// TwinCAT 3 PLC project SmartLogisticsBasic
// ProgramVersion: 3.1.4026.16
// libraries:
//   Tc2_BA, * (Beckhoff Automation GmbH)
//   Tc2_BABasic, * (Beckhoff Automation GmbH)
//   Tc2_BACnetRev12, * (Beckhoff Automation GmbH)
//   Tc2_CncBase, * (Beckhoff Automation GmbH)
//   Tc2_CncHli, * (Beckhoff Automation GmbH)
//   Tc2_CncPlcopenP1, * (Beckhoff Automation GmbH)
//   Tc2_CncPlcopenP4, * (Beckhoff Automation GmbH)
//   Tc2_ControllerToolbox, * (Beckhoff Automation GmbH)
//   Tc2_Coupler, * (Beckhoff Automation GmbH)
//   Tc2_DALI, * (Beckhoff Automation GmbH)
//   Tc2_Database, * (Beckhoff Automation GmbH)
//   Tc2_DataExchange, * (Beckhoff Automation GmbH)
//   Tc2_DMX, * (Beckhoff Automation GmbH)
//   Tc2_Drive, * (Beckhoff Automation GmbH)
//   Tc2_EIB, * (Beckhoff Automation GmbH)
//   Tc2_EnOcean, * (Beckhoff Automation GmbH)
//   Tc2_EtherCAT, * (Beckhoff Automation GmbH)
//   Tc2_EthernetIP, * (Beckhoff Automation GmbH)
//   Tc2_FTP, * (Beckhoff Automation GmbH)
//   Tc2_GENIbus, * (Beckhoff Automation GmbH)
//   Tc2_HVAC, * (Beckhoff Automation GmbH)
//   Tc2_IoFunctions, * (Beckhoff Automation GmbH)
//   Tc2_KL85xx, * (Beckhoff Automation GmbH)
//   Tc2_LON, * (Beckhoff Automation GmbH)
//   Tc2_Math, * (Beckhoff Automation GmbH)
//   Tc2_MBus, * (Beckhoff Automation GmbH)
//   Tc2_MC2, * (Beckhoff Automation GmbH)
//   Tc2_MC2_Camming, * (Beckhoff Automation GmbH)
//   Tc2_MC2_Drive, * (Beckhoff Automation GmbH)
//   Tc2_MC2_FlyingSaw, * (Beckhoff Automation GmbH)
//   Tc2_MC2_XFC, * (Beckhoff Automation GmbH)
//   Tc2_MDP, * (Beckhoff Automation GmbH)
//   Tc2_ModbusRTU, * (Beckhoff Automation GmbH)
//   Tc2_ModbusSrv, * (Beckhoff Automation GmbH)
//   Tc2_MPBus, * (Beckhoff Automation GmbH)
//   Tc2_NC, * (Beckhoff Automation GmbH)
//   Tc2_NcDrive, * (Beckhoff Automation GmbH)
//   Tc2_NcFifoAxes, * (Beckhoff Automation GmbH)
//   Tc2_NCI, * (Beckhoff Automation GmbH)
//   Tc2_NciXFC, * (Beckhoff Automation GmbH)
//   Tc2_PlcInterpolation, * (Beckhoff Automation GmbH)
//   Tc2_ProfinetDiag, * (Beckhoff Automation GmbH)
//   Tc2_RFID, * (Beckhoff Automation GmbH)
//   Tc2_S5S7Com, * (Beckhoff Automation GmbH)
//   Tc2_SerialCom, * (Beckhoff Automation GmbH)
//   Tc2_SMI, * (Beckhoff Automation GmbH)
//   Tc2_SMS, * (Beckhoff Automation GmbH)
//   Tc2_Smtp, * (Beckhoff Automation GmbH)
//   Tc2_SPA, * (Beckhoff Automation GmbH)
//   Tc2_Standard, * (Beckhoff Automation GmbH)
//   Tc2_System, * (Beckhoff Automation GmbH)
// project tree:
//   GVLs/ GVL_SimitSp.TcGVL, GVL_System.TcGVL (not stored)
//   / PlcTask.TcTTO
//   POUs/ FB_Chrono.TcPOU, FB_Conveyor.TcPOU (not stored), FB_ConvStatistic.TcPOU, FB_ConvSys.TcPOU, FB_FlPos.TcPOU, FB_MyUpCounter.TcPOU, FB_RunControl.TcPOU, FB_SpeedControl.TcPOU, FC_GetMaxLapTime.TcPOU, MAIN.TcPOU
// real-time tasks:
//   TASK PlcTask: cycle T#10ms, priority 20, ADS port 350
//   TASK OPC UA Virtual: cycle T#10ms, priority 35, ADS port 351
// I/O:
//   DEVICE Device 1 (OPC UA Virtual), AmsNetId 192.168.200.222.2.1
// variable links:
//   SmartLogisticsBasic Instance <-> Device 1 (OPC UA Virtual)/Siemens.Simit.OpcUaServer.OpcUaServerService
//     PlcTask Outputs/GVL_System.bWrite_Enable <-> Outputs/Control/Write Enable
//   SmartLogisticsBasic Instance <-> Device 1 (OPC UA Virtual)/Siemens.Simit.OpcUaServer.OpcUaServerService/urn:vmw11:Siemens:Simit.OpcUaServer.OPC UA Server/InSimitOpcBin/Ix_Enable
//     PlcTask Inputs/GVL_SimitSp.Ix_Enable <-> Inputs/Value
//   SmartLogisticsBasic Instance <-> Device 1 (OPC UA Virtual)/Siemens.Simit.OpcUaServer.OpcUaServerService/urn:vmw11:Siemens:Simit.OpcUaServer.OPC UA Server/InSimitOpcBin/Ix_LSensorBlue
//     PlcTask Inputs/GVL_SimitSp.Ix_LSensorBlue <-> Inputs/Value
//   SmartLogisticsBasic Instance <-> Device 1 (OPC UA Virtual)/Siemens.Simit.OpcUaServer.OpcUaServerService/urn:vmw11:Siemens:Simit.OpcUaServer.OPC UA Server/InSimitOpcBin/Ix_LSensorOrange
//     PlcTask Inputs/GVL_SimitSp.Ix_LSensorOrange <-> Inputs/Value
//   SmartLogisticsBasic Instance <-> Device 1 (OPC UA Virtual)/Siemens.Simit.OpcUaServer.OpcUaServerService/urn:vmw11:Siemens:Simit.OpcUaServer.OPC UA Server/InSimitOpcBin/Ix_LSensorPurple
//     PlcTask Inputs/GVL_SimitSp.Ix_LSensorPurple <-> Inputs/Value
//   SmartLogisticsBasic Instance <-> Device 1 (OPC UA Virtual)/Siemens.Simit.OpcUaServer.OpcUaServerService/urn:vmw11:Siemens:Simit.OpcUaServer.OPC UA Server/InSimitOpcBin/Ix_LSensorYellow
//     PlcTask Inputs/GVL_SimitSp.Ix_LSensorYellow <-> Inputs/Value
//   SmartLogisticsBasic Instance <-> Device 1 (OPC UA Virtual)/Siemens.Simit.OpcUaServer.OpcUaServerService/urn:vmw11:Siemens:Simit.OpcUaServer.OPC UA Server/InSimitOpcBin/Ix_Left
//     PlcTask Inputs/GVL_SimitSp.Ix_Left <-> Inputs/Value
//   SmartLogisticsBasic Instance <-> Device 1 (OPC UA Virtual)/Siemens.Simit.OpcUaServer.OpcUaServerService/urn:vmw11:Siemens:Simit.OpcUaServer.OPC UA Server/InSimitOpcBin/Ix_ManAuto
//     PlcTask Inputs/GVL_SimitSp.Ix_ManAuto <-> Inputs/Value
//   SmartLogisticsBasic Instance <-> Device 1 (OPC UA Virtual)/Siemens.Simit.OpcUaServer.OpcUaServerService/urn:vmw11:Siemens:Simit.OpcUaServer.OPC UA Server/InSimitOpcBin/Ix_NotAus
//     PlcTask Inputs/GVL_SimitSp.Ix_NotAus <-> Inputs/Value
//   SmartLogisticsBasic Instance <-> Device 1 (OPC UA Virtual)/Siemens.Simit.OpcUaServer.OpcUaServerService/urn:vmw11:Siemens:Simit.OpcUaServer.OPC UA Server/InSimitOpcBin/Ix_Off
//     PlcTask Inputs/GVL_SimitSp.Ix_Off <-> Inputs/Value
//   SmartLogisticsBasic Instance <-> Device 1 (OPC UA Virtual)/Siemens.Simit.OpcUaServer.OpcUaServerService/urn:vmw11:Siemens:Simit.OpcUaServer.OPC UA Server/InSimitOpcBin/Ix_On
//     PlcTask Inputs/GVL_SimitSp.Ix_On <-> Inputs/Value
//   SmartLogisticsBasic Instance <-> Device 1 (OPC UA Virtual)/Siemens.Simit.OpcUaServer.OpcUaServerService/urn:vmw11:Siemens:Simit.OpcUaServer.OPC UA Server/InSimitOpcBin/Ix_PowerOn
//     PlcTask Inputs/GVL_SimitSp.Ix_PowerOn <-> Inputs/Value
//   SmartLogisticsBasic Instance <-> Device 1 (OPC UA Virtual)/Siemens.Simit.OpcUaServer.OpcUaServerService/urn:vmw11:Siemens:Simit.OpcUaServer.OPC UA Server/InSimitOpcBin/Ix_RSensorBlue
//     PlcTask Inputs/GVL_SimitSp.Ix_RSensorBlue <-> Inputs/Value
//   SmartLogisticsBasic Instance <-> Device 1 (OPC UA Virtual)/Siemens.Simit.OpcUaServer.OpcUaServerService/urn:vmw11:Siemens:Simit.OpcUaServer.OPC UA Server/InSimitOpcBin/Ix_RSensorOrange
//     PlcTask Inputs/GVL_SimitSp.Ix_RSensorOrange <-> Inputs/Value
//   SmartLogisticsBasic Instance <-> Device 1 (OPC UA Virtual)/Siemens.Simit.OpcUaServer.OpcUaServerService/urn:vmw11:Siemens:Simit.OpcUaServer.OPC UA Server/InSimitOpcBin/Ix_RSensorPurple
//     PlcTask Inputs/GVL_SimitSp.Ix_RSensorPurple <-> Inputs/Value
//   SmartLogisticsBasic Instance <-> Device 1 (OPC UA Virtual)/Siemens.Simit.OpcUaServer.OpcUaServerService/urn:vmw11:Siemens:Simit.OpcUaServer.OPC UA Server/InSimitOpcBin/Ix_RSensorYellow
//     PlcTask Inputs/GVL_SimitSp.Ix_RSensorYellow <-> Inputs/Value
//   SmartLogisticsBasic Instance <-> Device 1 (OPC UA Virtual)/Siemens.Simit.OpcUaServer.OpcUaServerService/urn:vmw11:Siemens:Simit.OpcUaServer.OPC UA Server/InSimitOpcBin/Ix_Reset
//     PlcTask Inputs/GVL_SimitSp.Ix_Reset <-> Inputs/Value
//   SmartLogisticsBasic Instance <-> Device 1 (OPC UA Virtual)/Siemens.Simit.OpcUaServer.OpcUaServerService/urn:vmw11:Siemens:Simit.OpcUaServer.OPC UA Server/InSimitOpcBin/Ix_Right
//     PlcTask Inputs/GVL_SimitSp.Ix_Right <-> Inputs/Value
//   SmartLogisticsBasic Instance <-> Device 1 (OPC UA Virtual)/Siemens.Simit.OpcUaServer.OpcUaServerService/urn:vmw11:Siemens:Simit.OpcUaServer.OPC UA Server/InSimitOpcInt/Iw_SliderValue
//     PlcTask Inputs/GVL_SimitSp.Iw_SliderValue <-> Inputs/Value
//   SmartLogisticsBasic Instance <-> Device 1 (OPC UA Virtual)/Siemens.Simit.OpcUaServer.OpcUaServerService/urn:vmw11:Siemens:Simit.OpcUaServer.OPC UA Server/OutSimitOpcBin/Qx_EnableVarSpeedBlue
//     PlcTask Outputs/GVL_SimitSp.Qx_EnableVarSpeedBlue <-> Outputs/Value
//   SmartLogisticsBasic Instance <-> Device 1 (OPC UA Virtual)/Siemens.Simit.OpcUaServer.OpcUaServerService/urn:vmw11:Siemens:Simit.OpcUaServer.OPC UA Server/OutSimitOpcBin/Qx_EnableVarSpeedOrange
//     PlcTask Outputs/GVL_SimitSp.Qx_EnableVarSpeedOrange <-> Outputs/Value
//   SmartLogisticsBasic Instance <-> Device 1 (OPC UA Virtual)/Siemens.Simit.OpcUaServer.OpcUaServerService/urn:vmw11:Siemens:Simit.OpcUaServer.OPC UA Server/OutSimitOpcBin/Qx_EnableVarSpeedPurple
//     PlcTask Outputs/GVL_SimitSp.Qx_EnableVarSpeedPurple <-> Outputs/Value
//   SmartLogisticsBasic Instance <-> Device 1 (OPC UA Virtual)/Siemens.Simit.OpcUaServer.OpcUaServerService/urn:vmw11:Siemens:Simit.OpcUaServer.OPC UA Server/OutSimitOpcBin/Qx_EnableVarSpeedYellow
//     PlcTask Outputs/GVL_SimitSp.Qx_EnableVarSpeedYellow <-> Outputs/Value
//   SmartLogisticsBasic Instance <-> Device 1 (OPC UA Virtual)/Siemens.Simit.OpcUaServer.OpcUaServerService/urn:vmw11:Siemens:Simit.OpcUaServer.OPC UA Server/OutSimitOpcBin/Qx_FullSpeedBlue
//     PlcTask Outputs/GVL_SimitSp.Qx_FullSpeedBlue <-> Outputs/Value
//   SmartLogisticsBasic Instance <-> Device 1 (OPC UA Virtual)/Siemens.Simit.OpcUaServer.OpcUaServerService/urn:vmw11:Siemens:Simit.OpcUaServer.OPC UA Server/OutSimitOpcBin/Qx_FullSpeedOrange
//     PlcTask Outputs/GVL_SimitSp.Qx_FullSpeedOrange <-> Outputs/Value
//   SmartLogisticsBasic Instance <-> Device 1 (OPC UA Virtual)/Siemens.Simit.OpcUaServer.OpcUaServerService/urn:vmw11:Siemens:Simit.OpcUaServer.OPC UA Server/OutSimitOpcBin/Qx_FullSpeedPurple
//     PlcTask Outputs/GVL_SimitSp.Qx_FullSpeedPurple <-> Outputs/Value
//   SmartLogisticsBasic Instance <-> Device 1 (OPC UA Virtual)/Siemens.Simit.OpcUaServer.OpcUaServerService/urn:vmw11:Siemens:Simit.OpcUaServer.OPC UA Server/OutSimitOpcBin/Qx_FullSpeedYellow
//     PlcTask Outputs/GVL_SimitSp.Qx_FullSpeedYellow <-> Outputs/Value
//   SmartLogisticsBasic Instance <-> Device 1 (OPC UA Virtual)/Siemens.Simit.OpcUaServer.OpcUaServerService/urn:vmw11:Siemens:Simit.OpcUaServer.OPC UA Server/OutSimitOpcBin/Qx_MotorAcwBlue
//     PlcTask Outputs/GVL_SimitSp.Qx_MotorAcwBlue <-> Outputs/Value
//   SmartLogisticsBasic Instance <-> Device 1 (OPC UA Virtual)/Siemens.Simit.OpcUaServer.OpcUaServerService/urn:vmw11:Siemens:Simit.OpcUaServer.OPC UA Server/OutSimitOpcBin/Qx_MotorAcwOrange
//     PlcTask Outputs/GVL_SimitSp.Qx_MotorAcwOrange <-> Outputs/Value
//   SmartLogisticsBasic Instance <-> Device 1 (OPC UA Virtual)/Siemens.Simit.OpcUaServer.OpcUaServerService/urn:vmw11:Siemens:Simit.OpcUaServer.OPC UA Server/OutSimitOpcBin/Qx_MotorAcwPurple
//     PlcTask Outputs/GVL_SimitSp.Qx_MotorAcwPurple <-> Outputs/Value
//   SmartLogisticsBasic Instance <-> Device 1 (OPC UA Virtual)/Siemens.Simit.OpcUaServer.OpcUaServerService/urn:vmw11:Siemens:Simit.OpcUaServer.OPC UA Server/OutSimitOpcBin/Qx_MotorAcwYellow
//     PlcTask Outputs/GVL_SimitSp.Qx_MotorAcwYellow <-> Outputs/Value
//   SmartLogisticsBasic Instance <-> Device 1 (OPC UA Virtual)/Siemens.Simit.OpcUaServer.OpcUaServerService/urn:vmw11:Siemens:Simit.OpcUaServer.OPC UA Server/OutSimitOpcBin/Qx_MotorCwBlue
//     PlcTask Outputs/GVL_SimitSp.Qx_MotorCwBlue <-> Outputs/Value
//   SmartLogisticsBasic Instance <-> Device 1 (OPC UA Virtual)/Siemens.Simit.OpcUaServer.OpcUaServerService/urn:vmw11:Siemens:Simit.OpcUaServer.OPC UA Server/OutSimitOpcBin/Qx_MotorCwOrange
//     PlcTask Outputs/GVL_SimitSp.Qx_MotorCwOrange <-> Outputs/Value
//   SmartLogisticsBasic Instance <-> Device 1 (OPC UA Virtual)/Siemens.Simit.OpcUaServer.OpcUaServerService/urn:vmw11:Siemens:Simit.OpcUaServer.OPC UA Server/OutSimitOpcBin/Qx_MotorCwPurple
//     PlcTask Outputs/GVL_SimitSp.Qx_MotorCwPurple <-> Outputs/Value
//   SmartLogisticsBasic Instance <-> Device 1 (OPC UA Virtual)/Siemens.Simit.OpcUaServer.OpcUaServerService/urn:vmw11:Siemens:Simit.OpcUaServer.OPC UA Server/OutSimitOpcBin/Qx_MotorCwYellow
//     PlcTask Outputs/GVL_SimitSp.Qx_MotorCwYellow <-> Outputs/Value
//   SmartLogisticsBasic Instance <-> Device 1 (OPC UA Virtual)/Siemens.Simit.OpcUaServer.OpcUaServerService/urn:vmw11:Siemens:Simit.OpcUaServer.OPC UA Server/OutSimitOpcBin/Qx_StopperLeftBlue
//     PlcTask Outputs/GVL_SimitSp.Qx_StopperLeftBlue <-> Outputs/Value
//   SmartLogisticsBasic Instance <-> Device 1 (OPC UA Virtual)/Siemens.Simit.OpcUaServer.OpcUaServerService/urn:vmw11:Siemens:Simit.OpcUaServer.OPC UA Server/OutSimitOpcBin/Qx_StopperLeftOrange
//     PlcTask Outputs/GVL_SimitSp.Qx_StopperLeftOrange <-> Outputs/Value
//   SmartLogisticsBasic Instance <-> Device 1 (OPC UA Virtual)/Siemens.Simit.OpcUaServer.OpcUaServerService/urn:vmw11:Siemens:Simit.OpcUaServer.OPC UA Server/OutSimitOpcBin/Qx_StopperLeftPurble
//     PlcTask Outputs/GVL_SimitSp.Qx_StopperLeftPurble <-> Outputs/Value
//   SmartLogisticsBasic Instance <-> Device 1 (OPC UA Virtual)/Siemens.Simit.OpcUaServer.OpcUaServerService/urn:vmw11:Siemens:Simit.OpcUaServer.OPC UA Server/OutSimitOpcBin/Qx_StopperLeftYellow
//     PlcTask Outputs/GVL_SimitSp.Qx_StopperLeftYellow <-> Outputs/Value
//   SmartLogisticsBasic Instance <-> Device 1 (OPC UA Virtual)/Siemens.Simit.OpcUaServer.OpcUaServerService/urn:vmw11:Siemens:Simit.OpcUaServer.OPC UA Server/OutSimitOpcBin/Qx_StopperRightBlue
//     PlcTask Outputs/GVL_SimitSp.Qx_StopperRightBlue <-> Outputs/Value
//   SmartLogisticsBasic Instance <-> Device 1 (OPC UA Virtual)/Siemens.Simit.OpcUaServer.OpcUaServerService/urn:vmw11:Siemens:Simit.OpcUaServer.OPC UA Server/OutSimitOpcBin/Qx_StopperRightOrange
//     PlcTask Outputs/GVL_SimitSp.Qx_StopperRightOrange <-> Outputs/Value
//   SmartLogisticsBasic Instance <-> Device 1 (OPC UA Virtual)/Siemens.Simit.OpcUaServer.OpcUaServerService/urn:vmw11:Siemens:Simit.OpcUaServer.OPC UA Server/OutSimitOpcBin/Qx_StopperRightPurble
//     PlcTask Outputs/GVL_SimitSp.Qx_StopperRightPurble <-> Outputs/Value
//   SmartLogisticsBasic Instance <-> Device 1 (OPC UA Virtual)/Siemens.Simit.OpcUaServer.OpcUaServerService/urn:vmw11:Siemens:Simit.OpcUaServer.OPC UA Server/OutSimitOpcBin/Qx_StopperRightYellow
//     PlcTask Outputs/GVL_SimitSp.Qx_StopperRightYellow <-> Outputs/Value
//   SmartLogisticsBasic Instance <-> Device 1 (OPC UA Virtual)/Siemens.Simit.OpcUaServer.OpcUaServerService/urn:vmw11:Siemens:Simit.OpcUaServer.OPC UA Server/OutSimitOpcInt/Qw_VarSpeedBlue
//     PlcTask Outputs/GVL_SimitSp.Qw_VarSpeedBlue <-> Outputs/Value
//   SmartLogisticsBasic Instance <-> Device 1 (OPC UA Virtual)/Siemens.Simit.OpcUaServer.OpcUaServerService/urn:vmw11:Siemens:Simit.OpcUaServer.OPC UA Server/OutSimitOpcInt/Qw_VarSpeedOrange
//     PlcTask Outputs/GVL_SimitSp.Qw_VarSpeedOrange <-> Outputs/Value
//   SmartLogisticsBasic Instance <-> Device 1 (OPC UA Virtual)/Siemens.Simit.OpcUaServer.OpcUaServerService/urn:vmw11:Siemens:Simit.OpcUaServer.OPC UA Server/OutSimitOpcInt/Qw_VarSpeedPurple
//     PlcTask Outputs/GVL_SimitSp.Qw_VarSpeedPurple <-> Outputs/Value
//   SmartLogisticsBasic Instance <-> Device 1 (OPC UA Virtual)/Siemens.Simit.OpcUaServer.OpcUaServerService/urn:vmw11:Siemens:Simit.OpcUaServer.OPC UA Server/OutSimitOpcInt/Qw_VarSpeedYellow
//     PlcTask Outputs/GVL_SimitSp.Qw_VarSpeedYellow <-> Outputs/Value
//   SmartLogisticsBasic Instance <-> Device 1 (OPC UA Virtual)/Siemens.Simit.OpcUaServer.OpcUaServerService/urn:vmw11:Siemens:Simit.OpcUaServer.OPC UA Server/OutSimitOpcInt/nDisplays
//     PlcTask Outputs/GVL_SimitSp.Qb_74 <-> Outputs/Value @bit 16
//     PlcTask Outputs/GVL_SimitSp.Qb_75 <-> Outputs/Value @bit 24
//     PlcTask Outputs/GVL_SimitSp.Qw_Display <-> Outputs/Value
//   SmartLogisticsBasic Instance <-> Device 1 (OPC UA Virtual)/Siemens.Simit.OpcUaServer.OpcUaServerService/urn:vmw11:Siemens:Simit.OpcUaServer.OPC UA Server/OutSimitOpcInt/nLights
//     PlcTask Outputs/GVL_SimitSp.Qx_LightBlue <-> Outputs/Value @bit 3
//     PlcTask Outputs/GVL_SimitSp.Qx_LightGreen <-> Outputs/Value
//     PlcTask Outputs/GVL_SimitSp.Qx_LightRed <-> Outputs/Value @bit 2
//     PlcTask Outputs/GVL_SimitSp.Qx_LightYellow <-> Outputs/Value @bit 1

CONFIGURATION SmartLogisticsBasic
    RESOURCE PLC ON TwinCAT3
        TASK PlcTask(INTERVAL := T#10ms, PRIORITY := 20);
        PROGRAM MAIN WITH PlcTask : MAIN;
    END_RESOURCE
END_CONFIGURATION

// ---- GVLs/GVL_SimitSp.TcGVL
{attribute 'qualified_only'}
VAR_GLOBAL
    {attribute 'TcLinkTo' := 'TIID^Device 1 (OPC UA Virtual)^Siemens.Simit.OpcUaServer.OpcUaServerService^urn:vmw11:Siemens:Simit.OpcUaServer.OPC UA Server^InSimitOpcBin^Ix_Enable^Inputs^Value'}
    Ix_Enable AT %I* : BOOL;                // Taster Freigabe (variable Geschwindigkeit)
    {attribute 'TcLinkTo' := 'TIID^Device 1 (OPC UA Virtual)^Siemens.Simit.OpcUaServer.OpcUaServerService^urn:vmw11:Siemens:Simit.OpcUaServer.OPC UA Server^InSimitOpcBin^Ix_Left^Inputs^Value'}
    Ix_Left AT %I* : BOOL;                  // Taster links
    {attribute 'TcLinkTo' := 'TIID^Device 1 (OPC UA Virtual)^Siemens.Simit.OpcUaServer.OpcUaServerService^urn:vmw11:Siemens:Simit.OpcUaServer.OPC UA Server^InSimitOpcBin^Ix_LSensorBlue^Inputs^Value'}
    Ix_LSensorBlue AT %I* : BOOL;           // Linker Näherungssensor Band blau
    {attribute 'TcLinkTo' := 'TIID^Device 1 (OPC UA Virtual)^Siemens.Simit.OpcUaServer.OpcUaServerService^urn:vmw11:Siemens:Simit.OpcUaServer.OPC UA Server^InSimitOpcBin^Ix_LSensorOrange^Inputs^Value'}
    Ix_LSensorOrange AT %I* : BOOL;         // Linker Näherungssensor Band orange
    {attribute 'TcLinkTo' := 'TIID^Device 1 (OPC UA Virtual)^Siemens.Simit.OpcUaServer.OpcUaServerService^urn:vmw11:Siemens:Simit.OpcUaServer.OPC UA Server^InSimitOpcBin^Ix_LSensorPurple^Inputs^Value'}
    Ix_LSensorPurple AT %I* : BOOL;         // Linker Näherungssensor Band lila
    {attribute 'TcLinkTo' := 'TIID^Device 1 (OPC UA Virtual)^Siemens.Simit.OpcUaServer.OpcUaServerService^urn:vmw11:Siemens:Simit.OpcUaServer.OPC UA Server^InSimitOpcBin^Ix_LSensorYellow^Inputs^Value'}
    Ix_LSensorYellow AT %I* : BOOL;         // Linker Näherungssensor Band gelb
    {attribute 'TcLinkTo' := 'TIID^Device 1 (OPC UA Virtual)^Siemens.Simit.OpcUaServer.OpcUaServerService^urn:vmw11:Siemens:Simit.OpcUaServer.OPC UA Server^InSimitOpcBin^Ix_ManAuto^Inputs^Value'}
    Ix_ManAuto AT %I* : BOOL;               // Schalter manueller oder automatischer Betrieb (0=manuell)
    {attribute 'TcLinkTo' := 'TIID^Device 1 (OPC UA Virtual)^Siemens.Simit.OpcUaServer.OpcUaServerService^urn:vmw11:Siemens:Simit.OpcUaServer.OPC UA Server^InSimitOpcBin^Ix_NotAus^Inputs^Value'}
    Ix_NotAus AT %I* : BOOL;                // NotAus Schalter
    {attribute 'TcLinkTo' := 'TIID^Device 1 (OPC UA Virtual)^Siemens.Simit.OpcUaServer.OpcUaServerService^urn:vmw11:Siemens:Simit.OpcUaServer.OPC UA Server^InSimitOpcBin^Ix_Off^Inputs^Value'}
    Ix_Off AT %I* : BOOL;                   // Taster Aus
    {attribute 'TcLinkTo' := 'TIID^Device 1 (OPC UA Virtual)^Siemens.Simit.OpcUaServer.OpcUaServerService^urn:vmw11:Siemens:Simit.OpcUaServer.OPC UA Server^InSimitOpcBin^Ix_On^Inputs^Value'}
    Ix_On AT %I* : BOOL;                    // Taster Ein
    {attribute 'TcLinkTo' := 'TIID^Device 1 (OPC UA Virtual)^Siemens.Simit.OpcUaServer.OpcUaServerService^urn:vmw11:Siemens:Simit.OpcUaServer.OPC UA Server^InSimitOpcBin^Ix_PowerOn^Inputs^Value'}
    Ix_PowerOn AT %I* : BOOL;               // Hauptschalter
    {attribute 'TcLinkTo' := 'TIID^Device 1 (OPC UA Virtual)^Siemens.Simit.OpcUaServer.OpcUaServerService^urn:vmw11:Siemens:Simit.OpcUaServer.OPC UA Server^InSimitOpcBin^Ix_Reset^Inputs^Value'}
    Ix_Reset AT %I* : BOOL;                 // Taster Reset
    {attribute 'TcLinkTo' := 'TIID^Device 1 (OPC UA Virtual)^Siemens.Simit.OpcUaServer.OpcUaServerService^urn:vmw11:Siemens:Simit.OpcUaServer.OPC UA Server^InSimitOpcBin^Ix_Right^Inputs^Value'}
    Ix_Right AT %I* : BOOL;                 // Taster rechts
    {attribute 'TcLinkTo' := 'TIID^Device 1 (OPC UA Virtual)^Siemens.Simit.OpcUaServer.OpcUaServerService^urn:vmw11:Siemens:Simit.OpcUaServer.OPC UA Server^InSimitOpcBin^Ix_RSensorBlue^Inputs^Value'}
    Ix_RSensorBlue AT %I* : BOOL;           // Rechter Näherungssensor Band blau
    {attribute 'TcLinkTo' := 'TIID^Device 1 (OPC UA Virtual)^Siemens.Simit.OpcUaServer.OpcUaServerService^urn:vmw11:Siemens:Simit.OpcUaServer.OPC UA Server^InSimitOpcBin^Ix_RSensorOrange^Inputs^Value'}
    Ix_RSensorOrange AT %I* : BOOL;         // Rechter Näherungssensor Band orange
    {attribute 'TcLinkTo' := 'TIID^Device 1 (OPC UA Virtual)^Siemens.Simit.OpcUaServer.OpcUaServerService^urn:vmw11:Siemens:Simit.OpcUaServer.OPC UA Server^InSimitOpcBin^Ix_RSensorPurple^Inputs^Value'}
    Ix_RSensorPurple AT %I* : BOOL;         // Rechter Näherungssensor Band lila
    {attribute 'TcLinkTo' := 'TIID^Device 1 (OPC UA Virtual)^Siemens.Simit.OpcUaServer.OpcUaServerService^urn:vmw11:Siemens:Simit.OpcUaServer.OPC UA Server^InSimitOpcBin^Ix_RSensorYellow^Inputs^Value'}
    Ix_RSensorYellow AT %I* : BOOL;         // Rechter Näherungssensor Band gelb

    {attribute 'TcLinkToOSO' := '<0,16,0>TIID^Device 1 (OPC UA Virtual)^Siemens.Simit.OpcUaServer.OpcUaServerService^urn:vmw11:Siemens:Simit.OpcUaServer.OPC UA Server^InSimitOpcInt^Iw_SliderValue^Inputs^Value'}
    Iw_SliderValue AT %I* : WORD;           // Schieber für variablen Eingabewert

    {attribute 'TcLinkTo' := 'TIID^Device 1 (OPC UA Virtual)^Siemens.Simit.OpcUaServer.OpcUaServerService^urn:vmw11:Siemens:Simit.OpcUaServer.OPC UA Server^OutSimitOpcBin^Qx_EnableVarSpeedBlue^Outputs^Value'}
    Qx_EnableVarSpeedBlue AT %Q* : BOOL;    // Freigabe der variablen Geschwindigkeit Band blau
    {attribute 'TcLinkTo' := 'TIID^Device 1 (OPC UA Virtual)^Siemens.Simit.OpcUaServer.OpcUaServerService^urn:vmw11:Siemens:Simit.OpcUaServer.OPC UA Server^OutSimitOpcBin^Qx_EnableVarSpeedOrange^Outputs^Value'}
    Qx_EnableVarSpeedOrange AT %Q* : BOOL;  // Freigabe der variablen Geschwindigkeit Band orange
    {attribute 'TcLinkTo' := 'TIID^Device 1 (OPC UA Virtual)^Siemens.Simit.OpcUaServer.OpcUaServerService^urn:vmw11:Siemens:Simit.OpcUaServer.OPC UA Server^OutSimitOpcBin^Qx_EnableVarSpeedPurple^Outputs^Value'}
    Qx_EnableVarSpeedPurple AT %Q* : BOOL;  // Freigabe der variablen Geschwindigkeit Band lila
    {attribute 'TcLinkTo' := 'TIID^Device 1 (OPC UA Virtual)^Siemens.Simit.OpcUaServer.OpcUaServerService^urn:vmw11:Siemens:Simit.OpcUaServer.OPC UA Server^OutSimitOpcBin^Qx_EnableVarSpeedYellow^Outputs^Value'}
    Qx_EnableVarSpeedYellow AT %Q* : BOOL;  // Freigabe der variablen Geschwindigkeit Band gelb
    {attribute 'TcLinkTo' := 'TIID^Device 1 (OPC UA Virtual)^Siemens.Simit.OpcUaServer.OpcUaServerService^urn:vmw11:Siemens:Simit.OpcUaServer.OPC UA Server^OutSimitOpcBin^Qx_FullSpeedBlue^Outputs^Value'}
    Qx_FullSpeedBlue AT %Q* : BOOL;         // Eilgang Band blau
    {attribute 'TcLinkTo' := 'TIID^Device 1 (OPC UA Virtual)^Siemens.Simit.OpcUaServer.OpcUaServerService^urn:vmw11:Siemens:Simit.OpcUaServer.OPC UA Server^OutSimitOpcBin^Qx_FullSpeedOrange^Outputs^Value'}
    Qx_FullSpeedOrange AT %Q* : BOOL;       // Eilgang Band orange
    {attribute 'TcLinkTo' := 'TIID^Device 1 (OPC UA Virtual)^Siemens.Simit.OpcUaServer.OpcUaServerService^urn:vmw11:Siemens:Simit.OpcUaServer.OPC UA Server^OutSimitOpcBin^Qx_FullSpeedPurple^Outputs^Value'}
    Qx_FullSpeedPurple AT %Q* : BOOL;       // Eilgang Band lila
    {attribute 'TcLinkTo' := 'TIID^Device 1 (OPC UA Virtual)^Siemens.Simit.OpcUaServer.OpcUaServerService^urn:vmw11:Siemens:Simit.OpcUaServer.OPC UA Server^OutSimitOpcBin^Qx_FullSpeedYellow^Outputs^Value'}
    Qx_FullSpeedYellow AT %Q* : BOOL;       // Eilgang Band gelb
    {attribute 'TcLinkToOSO' := '<0,1,3>TIID^Device 1 (OPC UA Virtual)^Siemens.Simit.OpcUaServer.OpcUaServerService^urn:vmw11:Siemens:Simit.OpcUaServer.OPC UA Server^OutSimitOpcInt^nLights^Outputs^Value'}
    Qx_LightBlue AT %Q* : BOOL;             // Blaue Lampe
    {attribute 'TcLinkToOSO' := '<0,1,2>TIID^Device 1 (OPC UA Virtual)^Siemens.Simit.OpcUaServer.OpcUaServerService^urn:vmw11:Siemens:Simit.OpcUaServer.OPC UA Server^OutSimitOpcInt^nLights^Outputs^Value'}
    Qx_LightRed AT %Q* : BOOL;              // Rote Lampe
    {attribute 'TcLinkToOSO' := '<0,1,1>TIID^Device 1 (OPC UA Virtual)^Siemens.Simit.OpcUaServer.OpcUaServerService^urn:vmw11:Siemens:Simit.OpcUaServer.OPC UA Server^OutSimitOpcInt^nLights^Outputs^Value'}
    Qx_LightYellow AT %Q* : BOOL;           // Gelbe Lampe
    {attribute 'TcLinkToOSO' := '<0,1,0>TIID^Device 1 (OPC UA Virtual)^Siemens.Simit.OpcUaServer.OpcUaServerService^urn:vmw11:Siemens:Simit.OpcUaServer.OPC UA Server^OutSimitOpcInt^nLights^Outputs^Value'}
    Qx_LightGreen AT %Q* : BOOL;            // Grüne Lampe
    {attribute 'TcLinkTo' := 'TIID^Device 1 (OPC UA Virtual)^Siemens.Simit.OpcUaServer.OpcUaServerService^urn:vmw11:Siemens:Simit.OpcUaServer.OPC UA Server^OutSimitOpcBin^Qx_MotorAcwBlue^Outputs^Value'}
    Qx_MotorAcwBlue AT %Q* : BOOL;          // Motor dreht nach rechts (Gegenuhrzeigersinn Acw) Band blau
    {attribute 'TcLinkTo' := 'TIID^Device 1 (OPC UA Virtual)^Siemens.Simit.OpcUaServer.OpcUaServerService^urn:vmw11:Siemens:Simit.OpcUaServer.OPC UA Server^OutSimitOpcBin^Qx_MotorAcwOrange^Outputs^Value'}
    Qx_MotorAcwOrange AT %Q* : BOOL;        // Motor dreht nach rechts (Gegenuhrzeigersinn Acw) Band orange
    {attribute 'TcLinkTo' := 'TIID^Device 1 (OPC UA Virtual)^Siemens.Simit.OpcUaServer.OpcUaServerService^urn:vmw11:Siemens:Simit.OpcUaServer.OPC UA Server^OutSimitOpcBin^Qx_MotorAcwPurple^Outputs^Value'}
    Qx_MotorAcwPurple AT %Q* : BOOL;        // Motor dreht nach rechts (Gegenuhrzeigersinn Acw) Band lila
    {attribute 'TcLinkTo' := 'TIID^Device 1 (OPC UA Virtual)^Siemens.Simit.OpcUaServer.OpcUaServerService^urn:vmw11:Siemens:Simit.OpcUaServer.OPC UA Server^OutSimitOpcBin^Qx_MotorAcwYellow^Outputs^Value'}
    Qx_MotorAcwYellow AT %Q* : BOOL;        // Motor dreht nach rechts (Gegenuhrzeigersinn Acw) Band gelb
    {attribute 'TcLinkTo' := 'TIID^Device 1 (OPC UA Virtual)^Siemens.Simit.OpcUaServer.OpcUaServerService^urn:vmw11:Siemens:Simit.OpcUaServer.OPC UA Server^OutSimitOpcBin^Qx_MotorCwBlue^Outputs^Value'}
    Qx_MotorCwBlue AT %Q* : BOOL;           // Motor dreht nach links (Uhrzeigersinn Cw) Band blau
    {attribute 'TcLinkTo' := 'TIID^Device 1 (OPC UA Virtual)^Siemens.Simit.OpcUaServer.OpcUaServerService^urn:vmw11:Siemens:Simit.OpcUaServer.OPC UA Server^OutSimitOpcBin^Qx_MotorCwOrange^Outputs^Value'}
    Qx_MotorCwOrange AT %Q* : BOOL;         // Motor dreht nach links (Uhrzeigersinn Cw) Band orange
    {attribute 'TcLinkTo' := 'TIID^Device 1 (OPC UA Virtual)^Siemens.Simit.OpcUaServer.OpcUaServerService^urn:vmw11:Siemens:Simit.OpcUaServer.OPC UA Server^OutSimitOpcBin^Qx_MotorCwPurple^Outputs^Value'}
    Qx_MotorCwPurple AT %Q* : BOOL;         // Motor dreht nach links (Uhrzeigersinn Cw) Band lila
    {attribute 'TcLinkTo' := 'TIID^Device 1 (OPC UA Virtual)^Siemens.Simit.OpcUaServer.OpcUaServerService^urn:vmw11:Siemens:Simit.OpcUaServer.OPC UA Server^OutSimitOpcBin^Qx_MotorCwYellow^Outputs^Value'}
    Qx_MotorCwYellow AT %Q* : BOOL;         // Motor dreht nach links (Uhrzeigersinn Cw) Band gelb
    {attribute 'TcLinkTo' := 'TIID^Device 1 (OPC UA Virtual)^Siemens.Simit.OpcUaServer.OpcUaServerService^urn:vmw11:Siemens:Simit.OpcUaServer.OPC UA Server^OutSimitOpcBin^Qx_StopperLeftBlue^Outputs^Value'}
    Qx_StopperLeftBlue AT %Q* : BOOL;       // Stopper Blau Links
    {attribute 'TcLinkTo' := 'TIID^Device 1 (OPC UA Virtual)^Siemens.Simit.OpcUaServer.OpcUaServerService^urn:vmw11:Siemens:Simit.OpcUaServer.OPC UA Server^OutSimitOpcBin^Qx_StopperLeftOrange^Outputs^Value'}
    Qx_StopperLeftOrange AT %Q* : BOOL;     // Stopper Orange Links
    {attribute 'TcLinkTo' := 'TIID^Device 1 (OPC UA Virtual)^Siemens.Simit.OpcUaServer.OpcUaServerService^urn:vmw11:Siemens:Simit.OpcUaServer.OPC UA Server^OutSimitOpcBin^Qx_StopperLeftPurble^Outputs^Value'}
    Qx_StopperLeftPurble AT %Q* : BOOL;     // Stopper Violette Links
    {attribute 'TcLinkTo' := 'TIID^Device 1 (OPC UA Virtual)^Siemens.Simit.OpcUaServer.OpcUaServerService^urn:vmw11:Siemens:Simit.OpcUaServer.OPC UA Server^OutSimitOpcBin^Qx_StopperLeftYellow^Outputs^Value'}
    Qx_StopperLeftYellow AT %Q* : BOOL;     // Stopper Gelb Links
    {attribute 'TcLinkTo' := 'TIID^Device 1 (OPC UA Virtual)^Siemens.Simit.OpcUaServer.OpcUaServerService^urn:vmw11:Siemens:Simit.OpcUaServer.OPC UA Server^OutSimitOpcBin^Qx_StopperRightBlue^Outputs^Value'}
    Qx_StopperRightBlue AT %Q* : BOOL;      // Stopper Blau Rechts
    {attribute 'TcLinkTo' := 'TIID^Device 1 (OPC UA Virtual)^Siemens.Simit.OpcUaServer.OpcUaServerService^urn:vmw11:Siemens:Simit.OpcUaServer.OPC UA Server^OutSimitOpcBin^Qx_StopperRightOrange^Outputs^Value'}
    Qx_StopperRightOrange AT %Q* : BOOL;    // Stopper Orange Rechts
    {attribute 'TcLinkTo' := 'TIID^Device 1 (OPC UA Virtual)^Siemens.Simit.OpcUaServer.OpcUaServerService^urn:vmw11:Siemens:Simit.OpcUaServer.OPC UA Server^OutSimitOpcBin^Qx_StopperRightPurble^Outputs^Value'}
    Qx_StopperRightPurble AT %Q* : BOOL;    // Stopper Violette Rechts
    {attribute 'TcLinkTo' := 'TIID^Device 1 (OPC UA Virtual)^Siemens.Simit.OpcUaServer.OpcUaServerService^urn:vmw11:Siemens:Simit.OpcUaServer.OPC UA Server^OutSimitOpcBin^Qx_StopperRightYellow^Outputs^Value'}
    Qx_StopperRightYellow AT %Q* : BOOL;    // Stopper Gelb Rechts

    {attribute 'TcLinkToOSO' := '<0,16,0>TIID^Device 1 (OPC UA Virtual)^Siemens.Simit.OpcUaServer.OpcUaServerService^urn:vmw11:Siemens:Simit.OpcUaServer.OPC UA Server^OutSimitOpcInt^nDisplays^Outputs^Value'}
    Qw_Display AT %Q* : WORD;               // Anzeige für Ausgabewert
    {attribute 'TcLinkToOSO' := '<0,16,0>TIID^Device 1 (OPC UA Virtual)^Siemens.Simit.OpcUaServer.OpcUaServerService^urn:vmw11:Siemens:Simit.OpcUaServer.OPC UA Server^OutSimitOpcInt^Qw_VarSpeedBlue^Outputs^Value'}
    Qw_VarSpeedBlue AT %Q* : WORD;          // Variable Geschwindigkeitsvorgabe Band blue
    {attribute 'TcLinkToOSO' := '<0,16,0>TIID^Device 1 (OPC UA Virtual)^Siemens.Simit.OpcUaServer.OpcUaServerService^urn:vmw11:Siemens:Simit.OpcUaServer.OPC UA Server^OutSimitOpcInt^Qw_VarSpeedOrange^Outputs^Value'}
    Qw_VarSpeedOrange AT %Q* : WORD;        // Variable Geschwindigkeitsvorgabe Band orange
    {attribute 'TcLinkToOSO' := '<0,16,0>TIID^Device 1 (OPC UA Virtual)^Siemens.Simit.OpcUaServer.OpcUaServerService^urn:vmw11:Siemens:Simit.OpcUaServer.OPC UA Server^OutSimitOpcInt^Qw_VarSpeedPurple^Outputs^Value'}
    Qw_VarSpeedPurple AT %Q* : WORD;        // Variable Geschwindigkeitsvorgabe Band lila
    {attribute 'TcLinkToOSO' := '<0,16,0>TIID^Device 1 (OPC UA Virtual)^Siemens.Simit.OpcUaServer.OpcUaServerService^urn:vmw11:Siemens:Simit.OpcUaServer.OPC UA Server^OutSimitOpcInt^Qw_VarSpeedYellow^Outputs^Value'}
    Qw_VarSpeedYellow AT %Q* : WORD;        // Variable Geschwindigkeitsvorgabe Band yellow
	{attribute 'TcLinkToOSO' := '<0,8,16>TIID^Device 1 (OPC UA Virtual)^Siemens.Simit.OpcUaServer.OpcUaServerService^urn:vmw11:Siemens:Simit.OpcUaServer.OPC UA Server^OutSimitOpcInt^nDisplays^Outputs^Value'}
    Qb_74 AT %Q* : BYTE;                    // Anzeige für Ausgabewert Display links
    {attribute 'TcLinkToOSO' := '<0,8,24>TIID^Device 1 (OPC UA Virtual)^Siemens.Simit.OpcUaServer.OpcUaServerService^urn:vmw11:Siemens:Simit.OpcUaServer.OPC UA Server^OutSimitOpcInt^nDisplays^Outputs^Value'}
    Qb_75 AT %Q* : BYTE;                    // Anzeige für Ausgabewert Display rechts

END_VAR

// ---- POUs/MAIN.TcPOU
// Main Program Sweep (Cycle)
PROGRAM MAIN
VAR_TEMP 
  OB1_EV_CLASS : Byte;   // Bits 0-3 = 1 (Coming event), Bits 4-7 = 1 (Event class 1)
  OB1_SCAN_1 : Byte;   // 1 (Cold restart scan 1 of OB 1), 3 (Scan 2-n of OB 1)
  OB1_PRIORITY : Byte;   // Priority of OB Execution
  OB1_OB_NUMBR : Byte;   // 1 (Organization block 1, OB1)
  OB1_RESERVED_1 : Byte;   // Reserved for system
  OB1_RESERVED_2 : Byte;   // Reserved for system
  OB1_PREV_CYCLE : Int;   // Cycle time of previous OB1 scan (milliseconds)
  OB1_MIN_CYCLE : Int;   // Minimum cycle time of OB1 (milliseconds)
  OB1_MAX_CYCLE : Int;   // Maximum cycle time of OB1 (milliseconds)
  OB1_DATE_TIME : DATE_AND_TIME;   // Date and time OB1 started
END_VAR
VAR
  fbConvSys : FB_ConvSys;
END_VAR

fbConvSys();

END_PROGRAM

// ---- POUs/FB_ConvSys.TcPOU
// Bandrundlauf-Controller
// Kontrolliert den Bandrundlauf, ist eigentlich der Hauptbaustein(deshalb wird direkt auf PLC-Variablen zugegriffen(ohne Schnittstellenübergabe)
FUNCTION_BLOCK FB_ConvSys
VAR
    vsFB_ConvPurple : FB_Conveyor;
    vsFB_ConvOrange : FB_Conveyor;
    vsFB_ConvYellow : FB_Conveyor;
    vsFB_ConvBlue : FB_Conveyor;
	vsFB_CounterR: CTU := (PV:=0);
	FB_MyUpCounterL: FB_MyUpCounter;
	vsFB_FiPos: FB_FlPos;
	vsFB_Chrono: FB_Chrono;
	vsFB_ConvStatistic: FB_ConvStatistic;
	ix_LSensorPurpleLast: BOOL;
END_VAR
VAR_TEMP
	vti_CountValueL: INT;
	vtx_FlPosLap: BOOL;
	vtt_LapTime: TIME;
END_VAR
VAR_STAT
	vsi_Step: INT;
END_VAR

//Abbruch des Schrittkettenmodus
	IF GVL_SimitSp.Ix_Reset THEN
		vsi_Step:=000;
	END_IF

CASE vsi_Step OF
	
{region "init"}
	
	000: 	//Init-Modus
		GVL_SimitSp.Qx_MotorAcwPurple	:= FALSE;
		GVL_SimitSp.Qx_MotorCwPurple	:= FALSE;
		GVL_SimitSp.Qx_FullSpeedPurple	:= FALSE;
		GVL_SimitSp.Qx_MotorAcwOrange	:= FALSE;
		GVL_SimitSp.Qx_MotorCwOrange	:= FALSE;
		GVL_SimitSp.Qx_FullSpeedOrange	:= FALSE;
		GVL_SimitSp.Qx_MotorAcwYellow	:= FALSE;
		GVL_SimitSp.Qx_MotorCwYellow	:= FALSE;
		GVL_SimitSp.Qx_FullSpeedYellow	:= FALSE;
		GVL_SimitSp.Qx_MotorAcwBlue		:= FALSE;
		GVL_SimitSp.Qx_MotorCwBlue		:= FALSE;
		GVL_SimitSp.Qx_FullSpeedBlue	:= FALSE;
		GVL_SimitSp.Qx_LightGreen		:= FALSE;
	
		vsi_Step:=010;
	
{endregion}

	010: //Normalmodus
		vsFB_ConvPurple.vix_Left	:= GVL_SimitSp.Ix_Left;
		vsFB_ConvPurple.vix_Right	:= GVL_SimitSp.Ix_Right;
		vsFB_ConvOrange.vix_Left	:= GVL_SimitSp.Ix_Left;
		vsFB_ConvOrange.vix_Right	:= GVL_SimitSp.Ix_Right;
		vsFB_ConvYellow.vix_Left	:= GVL_SimitSp.Ix_Left;
		vsFB_ConvYellow.vix_Right	:= GVL_SimitSp.Ix_Right;
		vsFB_ConvBlue.vix_Left		:= GVL_SimitSp.Ix_Left;
		vsFB_ConvBlue.vix_Right		:= GVL_SimitSp.Ix_Right;
	
	IF 	GVL_SimitSp.Ix_Enable THEN
		GVL_SimitSp.Qx_LightGreen := TRUE;
	
	vsi_Step := 90;
	END_IF
	
	090: //Init von Schrittkettenmodus                                                                                    
		vsFB_ConvPurple.vix_Left	:= FALSE;                                                                              
		vsFB_ConvPurple.vix_Right	:= TRUE;                                                                              
		vsFB_ConvOrange.vix_Left	:= FALSE;                                                                              
		vsFB_ConvOrange.vix_Right	:= TRUE;                                                                              
		vsFB_ConvYellow.vix_Left	:= FALSE;                                                                              
		vsFB_ConvYellow.vix_Right	:= TRUE;                                                                              
		vsFB_ConvBlue.vix_Left		:= FALSE;                                                                              
		vsFB_ConvBlue.vix_Right		:= TRUE;                                                                             
		
	vsi_Step:=100;		//Bedingungslos in den nächsten Schritt schalten
	
	100: //Start Schrittketten-Ablauf
	IF GVL_SimitSp.Ix_RSensorPurple THEN
		vsFB_ConvPurple.vix_Left	:=TRUE;
		vsFB_ConvPurple.vix_Right	:=FALSE;
		
		vsi_Step:=110;
	END_IF;

	110:
	IF GVL_SimitSp.Ix_LSensorPurple THEN
		vsFB_ConvPurple.vix_Left	:=FALSE;
		vsFB_ConvPurple.vix_Right	:=TRUE;	
		vsFB_ConvOrange.vix_Left	:=FALSE;
		vsFB_ConvOrange.vix_Right	:=TRUE;	
		
		vsi_Step:=120;
	END_IF	
	
	120:
	IF GVL_SimitSp.Ix_RSensorOrange THEN
		vsFB_ConvOrange.vix_Left	:=TRUE;
		vsFB_ConvOrange.vix_Right	:=FALSE;
		
		vsi_Step:=130;
		END_IF
		
	130:
	IF GVL_SimitSp.Ix_LSensorOrange THEN
		vsFB_ConvOrange.vix_Left	:=FALSE;
		vsFB_ConvOrange.vix_Right	:=TRUE;
		vsFB_ConvYellow.vix_Left	:=FALSE;
		vsFB_ConvYellow.vix_Right	:=TRUE;
		
		vsi_Step:=140;
		END_IF
	
	140:
	IF GVL_SimitSp.Ix_RSensorYellow THEN
		vsFB_ConvYellow.vix_Left	:=TRUE;
		vsFB_ConvYellow.vix_Right	:=FALSE;
		
		vsi_Step:= 150;
		END_IF
		
	150:
	IF GVL_SimitSp.Ix_LSensorYellow THEN
		vsFB_ConvYellow.vix_Left	:=FALSE;
		vsFB_ConvYellow.vix_Right	:=TRUE;
		vsFB_ConvBlue.vix_Left	:=FALSE;
		vsFB_ConvBlue.vix_Right	:=TRUE;
		
		vsi_Step:= 160;
		END_IF
		
	160:
	IF GVL_SimitSp.Ix_RSensorBlue THEN
		vsFB_ConvBlue.vix_Left	:=TRUE;
		vsFB_ConvBlue.vix_Right	:=FALSE;
		
		vsi_Step:=170;
		END_IF
		
	170:
	IF GVL_SimitSp.Ix_LSensorBlue THEN
		vsFB_ConvBlue.vix_Left	:=FALSE;
		vsFB_ConvBlue.vix_Right	:=TRUE;
		vsFB_ConvPurple.vix_Left	:=FALSE;
		vsFB_ConvPurple.vix_Right	:=TRUE;
		
		vsi_Step:= 100;
		END_IF
				
	ELSE 							//ELSE von CASE
		vsi_Step :=000; 			//INIT
END_CASE;

(*Multiinstanzaufruf von Band lila*)
vsFB_ConvPurple(vix_Power := GVL_SimitSp.Ix_PowerOn,
                vix_On := GVL_SimitSp.Ix_On,
                vix_Off := GVL_SimitSp.Ix_Off,
//                 vix_Left := GVL_SimitSp.Ix_Left,
//                 vix_Right := GVL_SimitSp.Ix_Right,
                vix_ManAuto := GVL_SimitSp.Ix_ManAuto,                             
                viw_Speed := GVL_SimitSp.Iw_SliderValue,
                vqx_MotorCw => GVL_SimitSp.Qx_MotorCwPurple,
                vqx_MotorAcw => GVL_SimitSp.Qx_MotorAcwPurple,              
                vqx_VarSpeed => GVL_SimitSp.Qx_EnableVarSpeedPurple,
                vqw_Speed => GVL_SimitSp.Qw_VarSpeedPurple);
(*Multiinstanzaufruf von Band orange*)
vsFB_ConvOrange(vix_Power := GVL_SimitSp.Ix_PowerOn,
                vix_On := GVL_SimitSp.Ix_On,
                vix_Off := GVL_SimitSp.Ix_Off,
//                 vix_Left := GVL_SimitSp.Ix_Left,
//                 vix_Right := GVL_SimitSp.Ix_Right,
                vix_ManAuto := GVL_SimitSp.Ix_ManAuto,                              
                viw_Speed := GVL_SimitSp.Iw_SliderValue,
                vqx_MotorCw => GVL_SimitSp.Qx_MotorCwOrange,
                vqx_MotorAcw => GVL_SimitSp.Qx_MotorAcwOrange,               
                vqx_VarSpeed => GVL_SimitSp.Qx_EnableVarSpeedOrange,
                vqw_Speed => GVL_SimitSp.Qw_VarSpeedOrange);
(*Multiinstanzaufruf von Band yellow*)
vsFB_ConvYellow(vix_Power := GVL_SimitSp.Ix_PowerOn,
                vix_On := GVL_SimitSp.Ix_On,
                vix_Off := GVL_SimitSp.Ix_Off,
//                 vix_Left := GVL_SimitSp.Ix_Left,
//                 vix_Right := GVL_SimitSp.Ix_Right,
                vix_ManAuto := GVL_SimitSp.Ix_ManAuto,                              
                viw_Speed := GVL_SimitSp.Iw_SliderValue,
                vqx_MotorCw => GVL_SimitSp.Qx_MotorCwYellow,
                vqx_MotorAcw => GVL_SimitSp.Qx_MotorAcwYellow,               
                vqx_VarSpeed => GVL_SimitSp.Qx_EnableVarSpeedYellow,
                vqw_Speed => GVL_SimitSp.Qw_VarSpeedYellow);
(*Multiinstanzaufruf von Band blue*)
vsFB_ConvBlue(vix_Power := GVL_SimitSp.Ix_PowerOn,
                vix_On := GVL_SimitSp.Ix_On,
                vix_Off := GVL_SimitSp.Ix_Off,
//                 vix_Left := GVL_SimitSp.Ix_Left,
//                 vix_Right := GVL_SimitSp.Ix_Right,
                vix_ManAuto := GVL_SimitSp.Ix_ManAuto,               
                viw_Speed := GVL_SimitSp.Iw_SliderValue,
                vqx_MotorCw => GVL_SimitSp.Qx_MotorCwBlue,
                vqx_MotorAcw => GVL_SimitSp.Qx_MotorAcwBlue,               
                vqx_VarSpeed => GVL_SimitSp.Qx_EnableVarSpeedBlue,
                vqw_Speed => GVL_SimitSp.Qw_VarSpeedBlue); 

(*Rundlauf Anzeigen*)
GVL_SimitSp.Qx_LightBlue := GVL_SimitSp.Qx_MotorAcwBlue;  (*Gegenuhrzeigersinn Kontrolleuchte*)
GVL_SimitSp.Qx_LightYellow := GVL_SimitSp.Qx_MotorCwBlue; (*Uhrzeigersinn Kontrolleuchte*)
GVL_SimitSp.Qw_Display := GVL_SimitSp.Qw_VarSpeedPurple;  (*aktuelle variable Geschwindigkeit*)

(*Eilgang auf Enable Taster*)
GVL_SimitSp.Qx_FullSpeedPurple := GVL_SimitSp.Ix_Enable;
GVL_SimitSp.Qx_FullSpeedOrange := GVL_SimitSp.Ix_Enable;
GVL_SimitSp.Qx_FullSpeedYellow := GVL_SimitSp.Ix_Enable;
GVL_SimitSp.Qx_FullSpeedBlue := GVL_SimitSp.Ix_Enable; 

//Rundenzähler Rechtslauf
vsFB_CounterR(CU:= GVL_SimitSp.Ix_RSensorPurple AND GVL_SimitSp.Qx_MotorAcwPurple);
GVL_SimitSp.Qb_75 := WORD_TO_BYTE(vsFB_CounterR.CV);

//Rundenzähler Linkslauf
FB_MyUpCounterL(CU:= GVL_SimitSp.Ix_LSensorPurple AND GVL_SimitSp.Qx_MotorCwPurple, CV=> vti_CountValueL);
GVL_SimitSp.Qb_74 := INT_TO_BYTE(vti_CountValueL);

vsFB_FiPos(vix_Sig := GVL_SimitSp.Ix_LSensorPurple, vqx_FlPos => vtx_FlPosLap);
IF vtx_FlPosLap THEN
	vsFB_Chrono(vqt_LapTime => vtt_LapTime);
END_IF

IF GVL_SimitSp.Ix_LSensorPurple AND NOT ix_LSensorPurpleLast THEN
	vsFB_ConvStatistic(vit_LapTime := vtt_LapTime);
END_IF
ix_LSensorPurpleLast := GVL_SimitSp.Ix_LSensorPurple;

END_FUNCTION_BLOCK

// ---- POUs/FB_MyUpCounter.TcPOU
FUNCTION_BLOCK FB_MyUpCounter		//Rundenzähler Linkslauf
VAR_INPUT
	CU: BOOL;						//Count Up Signal
END_VAR
VAR_OUTPUT
	CV: INT;						//Counter Value
END_VAR
VAR
END_VAR
VAR_STAT
	vsi_Counter: INT;				//Speicher für den aktuellen Zählerstand 
	vsx_LastCU: BOOL;				//Zwischenspeicher letzter CU-Zustand
END_VAR

IF vsx_LastCU=FALSE AND CU=TRUE THEN
vsi_Counter:= vsi_Counter +1;
END_IF;
CV:= vsi_Counter;
vsx_LastCU:= CU;

END_FUNCTION_BLOCK

// ---- POUs/FB_FlPos.TcPOU
FUNCTION_BLOCK FB_FlPos
VAR_INPUT
    vix_Sig : BOOL;
END_VAR
VAR_OUTPUT
    vqx_FlPos : BOOL;
END_VAR
VAR
    vsx_LastSig : BOOL;
END_VAR

vqx_FlPos := (vix_Sig = TRUE) AND (vsx_LastSig = FALSE);
vsx_LastSig := vix_Sig;

END_FUNCTION_BLOCK

// ---- POUs/FB_Chrono.TcPOU
FUNCTION_BLOCK FB_Chrono
VAR_INPUT
END_VAR
VAR_OUTPUT
	vqt_LapTime: TIME;						// absolut oder relativ vergangene Zeit
END_VAR
VAR
	vst_ActTime: DATE_AND_TIME;				// aktuelle Zeit
	vst_LastTime: DATE_AND_TIME;			// zuletzt gespeicherte Zeit
	fbSysTime: FB_BA_GetTime;				// Systemzeit CPU
END_VAR

fbSysTime(bEN := TRUE, dtSysTi => vst_ActTime);
vqt_LapTime := vst_ActTime - vst_LastTime;
vst_LastTime := vst_ActTime;

END_FUNCTION_BLOCK

// ---- POUs/FB_ConvStatistic.TcPOU
FUNCTION_BLOCK FB_ConvStatistic				// Speicher der letzten 10 Rundenzeiten
VAR_INPUT
	vit_LapTime: TIME;						// Input letzter Rundenzeit
END_VAR
VAR_OUTPUT
END_VAR
VAR
	vsi_InPos: INT := 1;					// Zuweisung in welchem Arraybereich die nächste Zeit gespeichert werden soll
	vtt_MaxTime: Time;
END_VAR
VAR_STAT
	vsat_Laps: ARRAY[0..10] OF TIME;		// Deklaration von 10 Speicherplätzen
END_VAR

vsat_Laps[vsi_InPos] := vit_LapTime;		
IF vsi_InPos >= 10 THEN						//falls Array voll, ältester Eintrag überschreiben
	vsi_InPos := 1;							//
ELSE
	vsi_InPos := vsi_InPos +1;				// ansonsten Array 1 hochzählen
END_IF

vtt_MaxTime := FC_GetMaxLapTime(viqat_Laps := vsat_Laps);

END_FUNCTION_BLOCK

// ---- POUs/FC_GetMaxLapTime.TcPOU
FUNCTION FC_GetMaxLapTime : TIME		// Ermittlung der längsten zwischengespeicherten Rundenzeit
VAR_INPUT
END_VAR
VAR
	vti_I: INT;
END_VAR
VAR_IN_OUT
	viqat_Laps: ARRAY[0..10] OF TIME; 		//Durchgangsparameter
END_VAR

viqat_Laps[0] := T#0MS;							//maximumspeicher löschen
FOR vti_I := 1 TO 10 BY 1 DO 					//iteriert durch alle Einträge
IF (viqat_Laps[vti_I] > viqat_Laps[0]) THEN		//vergleiche maximum
	viqat_Laps[0] := viqat_Laps[vti_I];			//neues maximum speichern
END_IF
END_FOR
FC_GetMaxLapTime := viqat_Laps[0];				//Maximum als Rückgabewert

END_FUNCTION

// ---- POUs/FB_RunControl.TcPOU
// Band Controller
// Kontrolliert die Bandsteuerung anhand der gewünschten Eingabe-Funktionen    
FUNCTION_BLOCK FB_RunControl
VAR_INPUT 
    vix_Power : BOOL; // Hauptschalter
    vix_On : BOOL; // Band ein
    vix_Off : BOOL; // Band aus
    vix_AutoMode : BOOL; // Manuell oder Auto-Modus
    vix_Left : BOOL; // Linkslauf
    vix_Right : BOOL; // Rechtslauf
END_VAR
VAR_OUTPUT 
    vqx_Left : BOOL; // Linkslauf
    vqx_Right : BOOL; // Rechtslauf
END_VAR
VAR 
    vsx_DirLeftRight : BOOL; // Bit für Laufrichtung
    vsx_Running : BOOL; // Bit für Bandstatus
END_VAR

(*Start-Bedingungen*)
IF vix_Power AND (vix_On OR vsx_Running) THEN (*Selbsthaltung*)
    vsx_Running := TRUE;
    vqx_Right := vsx_DirLeftRight;
    vqx_Left := NOT vsx_DirLeftRight;
    
    IF vix_AutoMode THEN    
        (*Automatikbetrieb*)
        IF vix_Left THEN
            vqx_Left := TRUE;
            vqx_Right := FALSE;
        END_IF;
        IF vix_Right THEN
            vqx_Right := TRUE;
            vqx_Left := FALSE;
        END_IF;
    ELSE           
        (*Tippbetrieb*)    
        vqx_Left := vix_Left;
        vqx_Right := vix_Right;   
    END_IF;
    vsx_DirLeftRight := vqx_Right;
END_IF;

(*Stop-Bedingungen*)
IF NOT vix_Off OR NOT vix_Power THEN  
    vsx_Running := FALSE;
    vqx_Right := FALSE;
    vqx_Left := FALSE;
END_IF;

END_FUNCTION_BLOCK

// ---- POUs/FB_SpeedControl.TcPOU
// variable Geschwindigkeits Kontrolle
FUNCTION_BLOCK FB_SpeedControl
VAR_INPUT 
    viw_Speed : WORD; // Eingabe Soll-Geschwindigkeit
END_VAR
VAR_OUTPUT 
    vqx_VarSpeed : BOOL; // Enable Band Variable Geschwindigkeit
    vqw_Speed : WORD; // Band Soll-Geschwindigkeit
END_VAR
VAR 
    vsw_LastSpeed : WORD; // Soll-Geschwindigkeit von letztem Zyklus
	vtd_CalcSpeed: DINT;
	vtr_ScaleSpeed: REAL;
	vtr_NormSpeed: REAL;
END_VAR
VAR CONSTANT
	MAXNORM: INT := 27648;
	MINNORM: INT := 0;
	MAXSCALE: REAL := 100;
	MINSCALE: REAL := 0;
END_VAR

vqx_VarSpeed := TRUE;
IF (viw_Speed <> vsw_LastSpeed) THEN
    (*falls sich die Soll-Geschwindigkeit änderte*)
    (*Geschwindigkeit von WORD-Bereich auf Analogwert-Max skalieren*)   
	
 	vtd_CalcSpeed:= ABS(WORD_TO_DINT(viw_Speed)); //Wert in Absolutzahl speichern
	
	vtr_ScaleSpeed:= (MAXSCALE - MINSCALE)/ MAXNORM * DINT_TO_REAL(vtd_CalcSpeed) + MINSCALE;
	vtr_NormSpeed:= (((vtr_ScaleSpeed - MINSCALE) / (MAXSCALE - MINSCALE)) * (MAXNORM - MINNORM)) + MINNORM;
	vqw_Speed := INT_TO_WORD(REAL_TO_INT(vtr_NormSpeed));
    
	vsw_LastSpeed := viw_Speed; (*aktuelle Speed abspeichern für nächsten Zyklus*)
END_IF;

END_FUNCTION_BLOCK
